Staubli VAL3: POINT.dtx

Trajectory tTraj
  [0]
    TrajectoryItem tSuper[3]
      [0]
        num distance
        num moveType = 1
        num nTime
        num nStop
        num nTcpAction
        string comment = "appro"
        bool toStop
        mdesc nom_speed = {tmax=300, rmax=9999, leave=30, reach=30}
        InstrItem iInstr[3]
          [0]
            string sType
            string sData
          [1]
            string sType
            string sData
          [2]
            string sType
            string sData
        num nMoveId
      [1]
        num distance = 2
        num moveType = 1
        num nTime
        num nStop
        num nTcpAction = 2
        string comment = "point"
        bool toStop = true
        mdesc nom_speed = {tmax=300, rmax=9999, leave=30, reach=30}
        InstrItem iInstr[3]
          [0]
            string sType
            string sData
          [1]
            string sType
            string sData
          [2]
            string sType
            string sData
        num nMoveId
      [2]
        num distance
        num moveType = 1
        num nTime
        num nStop
        num nTcpAction
        string comment = "depart"
        bool toStop
        mdesc nom_speed = {tmax=300, rmax=9999, leave=30, reach=30}
        InstrItem iInstr[3]
          [0]
            string sType
            string sData
          [1]
            string sType
            string sData
          [2]
            string sType
            string sData
        num nMoveId
    string sID = "POINT pose"
    num nId
public bool bMoveType[3]
  [0] = true
  [1] = true
public bool bStepping
bool bToSave
frame fSetFrame = {fatherId=world[0]}
mdesc mMdesc = {accel=10, vel=10, decel=10, blend=off}
string sInstruction
public string sItems
string sMenu[8]
  [5] = "Duplicate"
  [7] = "New"
string sTrajType = "POINT"
pointRx pToGo = {fatherId=world[0]}
frame fFather = {fatherId=world[0]}
string sItemCycle
TrajPoint pEditPoint
  [0]
    TrajPointItem tData[3]
      [0]
        TrajectoryItem tSuper
          [0]
            num distance
            num moveType
            num nTime
            num nStop
            num nTcpAction
            string comment
            bool toStop
            mdesc nom_speed = {vel=500, tmax=500, rmax=9999, leave=30, reach=30}
            InstrItem iInstr[3]
              [0]
                string sType
                string sData
              [1]
                string sType
                string sData
              [2]
                string sType
                string sData
            num nMoveId
        pointRx pPoint = {fatherId=pEditPoint[0].fFrame[0]}
        num nType
      [1]
        TrajectoryItem tSuper
          [0]
            num distance
            num moveType
            num nTime
            num nStop
            num nTcpAction
            string comment
            bool toStop
            mdesc nom_speed = {vel=500, tmax=500, rmax=9999, leave=30, reach=30}
            InstrItem iInstr[3]
              [0]
                string sType
                string sData
              [1]
                string sType
                string sData
              [2]
                string sType
                string sData
            num nMoveId
        pointRx pPoint = {fatherId=pEditPoint[0].fFrame[0]}
        num nType
      [2]
        TrajectoryItem tSuper
          [0]
            num distance
            num moveType
            num nTime
            num nStop
            num nTcpAction
            string comment
            bool toStop
            mdesc nom_speed = {vel=500, tmax=500, rmax=9999, leave=30, reach=30}
            InstrItem iInstr[3]
              [0]
                string sType
                string sData
              [1]
                string sType
                string sData
              [2]
                string sType
                string sData
            num nMoveId
        pointRx pPoint = {fatherId=pEditPoint[0].fFrame[0]}
        num nType
    frame fFrame = {fatherId=world[0]}
    num nIndexTool
    string sID
    num nIndexFrame
